{attribute 'GeneratedUsingTerminal: EK1122-0000-0018'}
{attribute addProperty BoxType "EK1122-0000-0018"}
{attribute addProperty Id "Beckhoff_CUxxxxsub_EK1100EK1100_1FC0878B2A_0001_CU1123_0000_0016A_0001_CU1123_0000_0016_30E128CC124"}
{attribute addProperty CRC "3191096088"}
{attribute addProperty Size "126"}
{attribute addProperty Name "Beckhoff CUxxxxEK1122"}
TYPE Beckhoff_CUxxxxEK1122_BE344318 EXTENDS EK1122_1FC0878B :
STRUCT
	{attribute addProperty Name "Beckhoff CUxxxxsub EK1100"}
	{attribute addProperty PreviousPort "Beckhoff CUxxxxEK1122 : D"}
	Beckhoff_CUxxxxsub_EK1100 : EK1100_1FC0878B;
	{attribute addProperty Name "A_0001(CU1123-0000-0016)"}
	{attribute addProperty PreviousPort "Beckhoff CUxxxxsub EK1100 : C"}
	A_0001_CU1123_0000_0016 : A_0001_CU1123_0000_0016_30E128CC;
END_STRUCT
END_TYPE

(* stored: Version 1.2.0.0, ProductVersion 3.1.4024.11
   DUT Beckhoff_CUxxxxEK1122_BE344318: Id {3c25ef2e-f619-425e-bb38-547b86299824} *)
